FUNCTION_BLOCK TEST_SEL (* Test IEC 61131-3 bit string SEL functions *)
  (* Standard: 61499-1 *)
  (* Version 0.0, 2006-09-03, JHC, Holobloc Inc *)
  (* Compiler header: package fb.rt.test; *)
  (* Compiler classdef: SimpleFB *)
  (* Compiler Java Sun JDK 1.5.0 *)
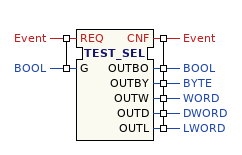
  EVENT_INPUT
    REQ WITH G; (* Normal Execution Request *)
  END_EVENT
  EVENT_OUTPUT
    CNF WITH OUTBO, OUTBY, OUTW, OUTD, OUTL; (* Execution Confirmation *)
  END_EVENT
  VAR_INPUT
    G : BOOL; (* Selection gate *)
  END_VAR
  VAR_OUTPUT
    OUTBO : BOOL; (* BOOL selection *)
    OUTBY : BYTE;
    OUTW : WORD;
    OUTD : DWORD;
    OUTL : LWORD;
  END_VAR
  ALGORITHM REQ IN FBD: (* Normally executed algorithm *)
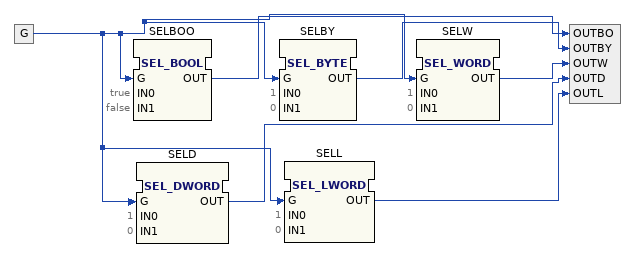
    FBS
      SELBOO : SEL_BOOL(IN0 := true, IN1 := false);
      SELBY : SEL_BYTE(IN0 := 1, IN1 := 0);
      SELW : SEL_WORD(IN0 := 1, IN1 := 0);
      SELD : SEL_DWORD(IN0 := 1, IN1 := 0);
      SELL : SEL_LWORD(IN0 := 1, IN1 := 0);
    END_FBS
    DATA_CONNECTIONS
      G TO SELBOO.G;
      SELBOO.OUT TO OUTBO;
      G TO SELBY.G;
      SELBY.OUT TO OUTBY;
      G TO SELW.G;
      SELW.OUT TO OUTW;
      G TO SELD.G;
      SELD.OUT TO OUTD;
      G TO SELL.G;
      SELL.OUT TO OUTL;
    END_CONNECTIONS
  END_ALGORITHM
END_FUNCTION_BLOCK
